// TIA Portal V19 export
TYPE "LEXCHANGETRAY_typeTrayParameter"
// stored: Access Published
   STRUCT
      specification { S7_SetPoint := 'True'} : Array[0..9] of "LEXCHANGETRAY_typeTraySpecification";   // 托盘规格
      selectSpecification { S7_SetPoint := 'True'} : Int;   // 选择规格
   END_STRUCT;
END_TYPE
